// TIA Portal V20 export
TYPE "LBP_typeTMMagazines"
TITLE = Tool management magazines / Magasins de gestion des outils
// User data type to store the magazine data / Type de données utilisateur pour l'enregistrement des données de magasin
   STRUCT
      MaxSpindleNumber : UInt;   // Maximum spindle number / Nombre maximal de broches
      NumberOfMagazines : UInt;   // Number of all magazines including loading and buffer magazines / Nombre total de magasins, y compris les magasins de chargement et de tampon
      Magazines : Array[1..64] of Struct   // All magazines including loading and buffer magazines / Tous les magasins, y compris les magasins de chargement et de tampon
         Number : UInt;   // Magazine number / Numéro de magasin
         "Type" : UInt;   // Magazine type / Type de magasin
         Places : UInt;   // Number of locations in magazine / Nombre d'emplacements dans le magasin
         TMNumber : UInt;   // Tool management number / Numéro de gestion des outils
      END_STRUCT;
   END_STRUCT;
   // // Magazines[2].Number : Magazine number / Numéro de magasin
   // // Magazines[3].Number : Magazine number / Numéro de magasin
   // // Magazines[4].Number : Magazine number / Numéro de magasin
   // // Magazines[5].Number : Magazine number / Numéro de magasin
   // // Magazines[6].Number : Magazine number / Numéro de magasin
   // // Magazines[7].Number : Magazine number / Numéro de magasin
   // // Magazines[8].Number : Magazine number / Numéro de magasin
   // // Magazines[9].Number : Magazine number / Numéro de magasin
   // // Magazines[10].Number : Magazine number / Numéro de magasin
   // // Magazines[11].Number : Magazine number / Numéro de magasin
   // // Magazines[12].Number : Magazine number / Numéro de magasin
   // // Magazines[13].Number : Magazine number / Numéro de magasin
   // // Magazines[14].Number : Magazine number / Numéro de magasin
   // // Magazines[15].Number : Magazine number / Numéro de magasin
   // // Magazines[16].Number : Magazine number / Numéro de magasin
   // // Magazines[17].Number : Magazine number / Numéro de magasin
   // // Magazines[18].Number : Magazine number / Numéro de magasin
   // // Magazines[19].Number : Magazine number / Numéro de magasin
   // // Magazines[20].Number : Magazine number / Numéro de magasin
   // // Magazines[21].Number : Magazine number / Numéro de magasin
   // // Magazines[22].Number : Magazine number / Numéro de magasin
   // // Magazines[23].Number : Magazine number / Numéro de magasin
   // // Magazines[24].Number : Magazine number / Numéro de magasin
   // // Magazines[25].Number : Magazine number / Numéro de magasin
   // // Magazines[26].Number : Magazine number / Numéro de magasin
   // // Magazines[27].Number : Magazine number / Numéro de magasin
   // // Magazines[28].Number : Magazine number / Numéro de magasin
   // // Magazines[29].Number : Magazine number / Numéro de magasin
   // // Magazines[30].Number : Magazine number / Numéro de magasin
   // // Magazines[31].Number : Magazine number / Numéro de magasin
   // // Magazines[32].Number : Magazine number / Numéro de magasin
   // // Magazines[33].Number : Magazine number / Numéro de magasin
   // // Magazines[34].Number : Magazine number / Numéro de magasin
   // // Magazines[35].Number : Magazine number / Numéro de magasin
   // // Magazines[36].Number : Magazine number / Numéro de magasin
   // // Magazines[37].Number : Magazine number / Numéro de magasin
   // // Magazines[38].Number : Magazine number / Numéro de magasin
   // // Magazines[39].Number : Magazine number / Numéro de magasin
   // // Magazines[40].Number : Magazine number / Numéro de magasin
   // // Magazines[41].Number : Magazine number / Numéro de magasin
   // // Magazines[42].Number : Magazine number / Numéro de magasin
   // // Magazines[43].Number : Magazine number / Numéro de magasin
   // // Magazines[44].Number : Magazine number / Numéro de magasin
   // // Magazines[45].Number : Magazine number / Numéro de magasin
   // // Magazines[46].Number : Magazine number / Numéro de magasin
   // // Magazines[47].Number : Magazine number / Numéro de magasin
   // // Magazines[48].Number : Magazine number / Numéro de magasin
   // // Magazines[49].Number : Magazine number / Numéro de magasin
   // // Magazines[50].Number : Magazine number / Numéro de magasin
   // // Magazines[51].Number : Magazine number / Numéro de magasin
   // // Magazines[52].Number : Magazine number / Numéro de magasin
   // // Magazines[53].Number : Magazine number / Numéro de magasin
   // // Magazines[54].Number : Magazine number / Numéro de magasin
   // // Magazines[55].Number : Magazine number / Numéro de magasin
   // // Magazines[56].Number : Magazine number / Numéro de magasin
   // // Magazines[57].Number : Magazine number / Numéro de magasin
   // // Magazines[58].Number : Magazine number / Numéro de magasin
   // // Magazines[59].Number : Magazine number / Numéro de magasin
   // // Magazines[60].Number : Magazine number / Numéro de magasin
   // // Magazines[61].Number : Magazine number / Numéro de magasin
   // // Magazines[62].Number : Magazine number / Numéro de magasin
   // // Magazines[63].Number : Magazine number / Numéro de magasin
   // // Magazines[64].Number : Magazine number / Numéro de magasin
   // // Magazines[2]."Type" : Magazine type / Type de magasin
   // // Magazines[3]."Type" : Magazine type / Type de magasin
   // // Magazines[4]."Type" : Magazine type / Type de magasin
   // // Magazines[5]."Type" : Magazine type / Type de magasin
   // // Magazines[6]."Type" : Magazine type / Type de magasin
   // // Magazines[7]."Type" : Magazine type / Type de magasin
   // // Magazines[8]."Type" : Magazine type / Type de magasin
   // // Magazines[9]."Type" : Magazine type / Type de magasin
   // // Magazines[10]."Type" : Magazine type / Type de magasin
   // // Magazines[11]."Type" : Magazine type / Type de magasin
   // // Magazines[12]."Type" : Magazine type / Type de magasin
   // // Magazines[13]."Type" : Magazine type / Type de magasin
   // // Magazines[14]."Type" : Magazine type / Type de magasin
   // // Magazines[15]."Type" : Magazine type / Type de magasin
   // // Magazines[16]."Type" : Magazine type / Type de magasin
   // // Magazines[17]."Type" : Magazine type / Type de magasin
   // // Magazines[18]."Type" : Magazine type / Type de magasin
   // // Magazines[19]."Type" : Magazine type / Type de magasin
   // // Magazines[20]."Type" : Magazine type / Type de magasin
   // // Magazines[21]."Type" : Magazine type / Type de magasin
   // // Magazines[22]."Type" : Magazine type / Type de magasin
   // // Magazines[23]."Type" : Magazine type / Type de magasin
   // // Magazines[24]."Type" : Magazine type / Type de magasin
   // // Magazines[25]."Type" : Magazine type / Type de magasin
   // // Magazines[26]."Type" : Magazine type / Type de magasin
   // // Magazines[27]."Type" : Magazine type / Type de magasin
   // // Magazines[28]."Type" : Magazine type / Type de magasin
   // // Magazines[29]."Type" : Magazine type / Type de magasin
   // // Magazines[30]."Type" : Magazine type / Type de magasin
   // // Magazines[31]."Type" : Magazine type / Type de magasin
   // // Magazines[32]."Type" : Magazine type / Type de magasin
   // // Magazines[33]."Type" : Magazine type / Type de magasin
   // // Magazines[34]."Type" : Magazine type / Type de magasin
   // // Magazines[35]."Type" : Magazine type / Type de magasin
   // // Magazines[36]."Type" : Magazine type / Type de magasin
   // // Magazines[37]."Type" : Magazine type / Type de magasin
   // // Magazines[38]."Type" : Magazine type / Type de magasin
   // // Magazines[39]."Type" : Magazine type / Type de magasin
   // // Magazines[40]."Type" : Magazine type / Type de magasin
   // // Magazines[41]."Type" : Magazine type / Type de magasin
   // // Magazines[42]."Type" : Magazine type / Type de magasin
   // // Magazines[43]."Type" : Magazine type / Type de magasin
   // // Magazines[44]."Type" : Magazine type / Type de magasin
   // // Magazines[45]."Type" : Magazine type / Type de magasin
   // // Magazines[46]."Type" : Magazine type / Type de magasin
   // // Magazines[47]."Type" : Magazine type / Type de magasin
   // // Magazines[48]."Type" : Magazine type / Type de magasin
   // // Magazines[49]."Type" : Magazine type / Type de magasin
   // // Magazines[50]."Type" : Magazine type / Type de magasin
   // // Magazines[51]."Type" : Magazine type / Type de magasin
   // // Magazines[52]."Type" : Magazine type / Type de magasin
   // // Magazines[53]."Type" : Magazine type / Type de magasin
   // // Magazines[54]."Type" : Magazine type / Type de magasin
   // // Magazines[55]."Type" : Magazine type / Type de magasin
   // // Magazines[56]."Type" : Magazine type / Type de magasin
   // // Magazines[57]."Type" : Magazine type / Type de magasin
   // // Magazines[58]."Type" : Magazine type / Type de magasin
   // // Magazines[59]."Type" : Magazine type / Type de magasin
   // // Magazines[60]."Type" : Magazine type / Type de magasin
   // // Magazines[61]."Type" : Magazine type / Type de magasin
   // // Magazines[62]."Type" : Magazine type / Type de magasin
   // // Magazines[63]."Type" : Magazine type / Type de magasin
   // // Magazines[64]."Type" : Magazine type / Type de magasin
   // // Magazines[2].Places : Number of locations in magazine / Nombre d'emplacements dans le magasin
   // // Magazines[3].Places : Number of locations in magazine / Nombre d'emplacements dans le magasin
   // // Magazines[4].Places : Number of locations in magazine / Nombre d'emplacements dans le magasin
   // // Magazines[5].Places : Number of locations in magazine / Nombre d'emplacements dans le magasin
   // // Magazines[6].Places : Number of locations in magazine / Nombre d'emplacements dans le magasin
   // // Magazines[7].Places : Number of locations in magazine / Nombre d'emplacements dans le magasin
   // // Magazines[8].Places : Number of locations in magazine / Nombre d'emplacements dans le magasin
   // // Magazines[9].Places : Number of locations in magazine / Nombre d'emplacements dans le magasin
   // // Magazines[10].Places : Number of locations in magazine / Nombre d'emplacements dans le magasin
   // // Magazines[11].Places : Number of locations in magazine / Nombre d'emplacements dans le magasin
   // // Magazines[12].Places : Number of locations in magazine / Nombre d'emplacements dans le magasin
   // // Magazines[13].Places : Number of locations in magazine / Nombre d'emplacements dans le magasin
   // // Magazines[14].Places : Number of locations in magazine / Nombre d'emplacements dans le magasin
   // // Magazines[15].Places : Number of locations in magazine / Nombre d'emplacements dans le magasin
   // // Magazines[16].Places : Number of locations in magazine / Nombre d'emplacements dans le magasin
   // // Magazines[17].Places : Number of locations in magazine / Nombre d'emplacements dans le magasin
   // // Magazines[18].Places : Number of locations in magazine / Nombre d'emplacements dans le magasin
   // // Magazines[19].Places : Number of locations in magazine / Nombre d'emplacements dans le magasin
   // // Magazines[20].Places : Number of locations in magazine / Nombre d'emplacements dans le magasin
   // // Magazines[21].Places : Number of locations in magazine / Nombre d'emplacements dans le magasin
   // // Magazines[22].Places : Number of locations in magazine / Nombre d'emplacements dans le magasin
   // // Magazines[23].Places : Number of locations in magazine / Nombre d'emplacements dans le magasin
   // // Magazines[24].Places : Number of locations in magazine / Nombre d'emplacements dans le magasin
   // // Magazines[25].Places : Number of locations in magazine / Nombre d'emplacements dans le magasin
   // // Magazines[26].Places : Number of locations in magazine / Nombre d'emplacements dans le magasin
   // // Magazines[27].Places : Number of locations in magazine / Nombre d'emplacements dans le magasin
   // // Magazines[28].Places : Number of locations in magazine / Nombre d'emplacements dans le magasin
   // // Magazines[29].Places : Number of locations in magazine / Nombre d'emplacements dans le magasin
   // // Magazines[30].Places : Number of locations in magazine / Nombre d'emplacements dans le magasin
   // // Magazines[31].Places : Number of locations in magazine / Nombre d'emplacements dans le magasin
   // // Magazines[32].Places : Number of locations in magazine / Nombre d'emplacements dans le magasin
   // // Magazines[33].Places : Number of locations in magazine / Nombre d'emplacements dans le magasin
   // // Magazines[34].Places : Number of locations in magazine / Nombre d'emplacements dans le magasin
   // // Magazines[35].Places : Number of locations in magazine / Nombre d'emplacements dans le magasin
   // // Magazines[36].Places : Number of locations in magazine / Nombre d'emplacements dans le magasin
   // // Magazines[37].Places : Number of locations in magazine / Nombre d'emplacements dans le magasin
   // // Magazines[38].Places : Number of locations in magazine / Nombre d'emplacements dans le magasin
   // // Magazines[39].Places : Number of locations in magazine / Nombre d'emplacements dans le magasin
   // // Magazines[40].Places : Number of locations in magazine / Nombre d'emplacements dans le magasin
   // // Magazines[41].Places : Number of locations in magazine / Nombre d'emplacements dans le magasin
   // // Magazines[42].Places : Number of locations in magazine / Nombre d'emplacements dans le magasin
   // // Magazines[43].Places : Number of locations in magazine / Nombre d'emplacements dans le magasin
   // // Magazines[44].Places : Number of locations in magazine / Nombre d'emplacements dans le magasin
   // // Magazines[45].Places : Number of locations in magazine / Nombre d'emplacements dans le magasin
   // // Magazines[46].Places : Number of locations in magazine / Nombre d'emplacements dans le magasin
   // // Magazines[47].Places : Number of locations in magazine / Nombre d'emplacements dans le magasin
   // // Magazines[48].Places : Number of locations in magazine / Nombre d'emplacements dans le magasin
   // // Magazines[49].Places : Number of locations in magazine / Nombre d'emplacements dans le magasin
   // // Magazines[50].Places : Number of locations in magazine / Nombre d'emplacements dans le magasin
   // // Magazines[51].Places : Number of locations in magazine / Nombre d'emplacements dans le magasin
   // // Magazines[52].Places : Number of locations in magazine / Nombre d'emplacements dans le magasin
   // // Magazines[53].Places : Number of locations in magazine / Nombre d'emplacements dans le magasin
   // // Magazines[54].Places : Number of locations in magazine / Nombre d'emplacements dans le magasin
   // // Magazines[55].Places : Number of locations in magazine / Nombre d'emplacements dans le magasin
   // // Magazines[56].Places : Number of locations in magazine / Nombre d'emplacements dans le magasin
   // // Magazines[57].Places : Number of locations in magazine / Nombre d'emplacements dans le magasin
   // // Magazines[58].Places : Number of locations in magazine / Nombre d'emplacements dans le magasin
   // // Magazines[59].Places : Number of locations in magazine / Nombre d'emplacements dans le magasin
   // // Magazines[60].Places : Number of locations in magazine / Nombre d'emplacements dans le magasin
   // // Magazines[61].Places : Number of locations in magazine / Nombre d'emplacements dans le magasin
   // // Magazines[62].Places : Number of locations in magazine / Nombre d'emplacements dans le magasin
   // // Magazines[63].Places : Number of locations in magazine / Nombre d'emplacements dans le magasin
   // // Magazines[64].Places : Number of locations in magazine / Nombre d'emplacements dans le magasin
   // // Magazines[2].TMNumber : Tool management number / Numéro de gestion des outils
   // // Magazines[3].TMNumber : Tool management number / Numéro de gestion des outils
   // // Magazines[4].TMNumber : Tool management number / Numéro de gestion des outils
   // // Magazines[5].TMNumber : Tool management number / Numéro de gestion des outils
   // // Magazines[6].TMNumber : Tool management number / Numéro de gestion des outils
   // // Magazines[7].TMNumber : Tool management number / Numéro de gestion des outils
   // // Magazines[8].TMNumber : Tool management number / Numéro de gestion des outils
   // // Magazines[9].TMNumber : Tool management number / Numéro de gestion des outils
   // // Magazines[10].TMNumber : Tool management number / Numéro de gestion des outils
   // // Magazines[11].TMNumber : Tool management number / Numéro de gestion des outils
   // // Magazines[12].TMNumber : Tool management number / Numéro de gestion des outils
   // // Magazines[13].TMNumber : Tool management number / Numéro de gestion des outils
   // // Magazines[14].TMNumber : Tool management number / Numéro de gestion des outils
   // // Magazines[15].TMNumber : Tool management number / Numéro de gestion des outils
   // // Magazines[16].TMNumber : Tool management number / Numéro de gestion des outils
   // // Magazines[17].TMNumber : Tool management number / Numéro de gestion des outils
   // // Magazines[18].TMNumber : Tool management number / Numéro de gestion des outils
   // // Magazines[19].TMNumber : Tool management number / Numéro de gestion des outils
   // // Magazines[20].TMNumber : Tool management number / Numéro de gestion des outils
   // // Magazines[21].TMNumber : Tool management number / Numéro de gestion des outils
   // // Magazines[22].TMNumber : Tool management number / Numéro de gestion des outils
   // // Magazines[23].TMNumber : Tool management number / Numéro de gestion des outils
   // // Magazines[24].TMNumber : Tool management number / Numéro de gestion des outils
   // // Magazines[25].TMNumber : Tool management number / Numéro de gestion des outils
   // // Magazines[26].TMNumber : Tool management number / Numéro de gestion des outils
   // // Magazines[27].TMNumber : Tool management number / Numéro de gestion des outils
   // // Magazines[28].TMNumber : Tool management number / Numéro de gestion des outils
   // // Magazines[29].TMNumber : Tool management number / Numéro de gestion des outils
   // // Magazines[30].TMNumber : Tool management number / Numéro de gestion des outils
   // // Magazines[31].TMNumber : Tool management number / Numéro de gestion des outils
   // // Magazines[32].TMNumber : Tool management number / Numéro de gestion des outils
   // // Magazines[33].TMNumber : Tool management number / Numéro de gestion des outils
   // // Magazines[34].TMNumber : Tool management number / Numéro de gestion des outils
   // // Magazines[35].TMNumber : Tool management number / Numéro de gestion des outils
   // // Magazines[36].TMNumber : Tool management number / Numéro de gestion des outils
   // // Magazines[37].TMNumber : Tool management number / Numéro de gestion des outils
   // // Magazines[38].TMNumber : Tool management number / Numéro de gestion des outils
   // // Magazines[39].TMNumber : Tool management number / Numéro de gestion des outils
   // // Magazines[40].TMNumber : Tool management number / Numéro de gestion des outils
   // // Magazines[41].TMNumber : Tool management number / Numéro de gestion des outils
   // // Magazines[42].TMNumber : Tool management number / Numéro de gestion des outils
   // // Magazines[43].TMNumber : Tool management number / Numéro de gestion des outils
   // // Magazines[44].TMNumber : Tool management number / Numéro de gestion des outils
   // // Magazines[45].TMNumber : Tool management number / Numéro de gestion des outils
   // // Magazines[46].TMNumber : Tool management number / Numéro de gestion des outils
   // // Magazines[47].TMNumber : Tool management number / Numéro de gestion des outils
   // // Magazines[48].TMNumber : Tool management number / Numéro de gestion des outils
   // // Magazines[49].TMNumber : Tool management number / Numéro de gestion des outils
   // // Magazines[50].TMNumber : Tool management number / Numéro de gestion des outils
   // // Magazines[51].TMNumber : Tool management number / Numéro de gestion des outils
   // // Magazines[52].TMNumber : Tool management number / Numéro de gestion des outils
   // // Magazines[53].TMNumber : Tool management number / Numéro de gestion des outils
   // // Magazines[54].TMNumber : Tool management number / Numéro de gestion des outils
   // // Magazines[55].TMNumber : Tool management number / Numéro de gestion des outils
   // // Magazines[56].TMNumber : Tool management number / Numéro de gestion des outils
   // // Magazines[57].TMNumber : Tool management number / Numéro de gestion des outils
   // // Magazines[58].TMNumber : Tool management number / Numéro de gestion des outils
   // // Magazines[59].TMNumber : Tool management number / Numéro de gestion des outils
   // // Magazines[60].TMNumber : Tool management number / Numéro de gestion des outils
   // // Magazines[61].TMNumber : Tool management number / Numéro de gestion des outils
   // // Magazines[62].TMNumber : Tool management number / Numéro de gestion des outils
   // // Magazines[63].TMNumber : Tool management number / Numéro de gestion des outils
   // // Magazines[64].TMNumber : Tool management number / Numéro de gestion des outils
   // // Magazines[1] : All magazines including loading and buffer magazines / Tous les magasins, y compris les magasins de chargement et de tampon
   // // Magazines[2] : All magazines including loading and buffer magazines / Tous les magasins, y compris les magasins de chargement et de tampon
   // // Magazines[3] : All magazines including loading and buffer magazines / Tous les magasins, y compris les magasins de chargement et de tampon
   // // Magazines[4] : All magazines including loading and buffer magazines / Tous les magasins, y compris les magasins de chargement et de tampon
   // // Magazines[5] : All magazines including loading and buffer magazines / Tous les magasins, y compris les magasins de chargement et de tampon
   // // Magazines[6] : All magazines including loading and buffer magazines / Tous les magasins, y compris les magasins de chargement et de tampon
   // // Magazines[7] : All magazines including loading and buffer magazines / Tous les magasins, y compris les magasins de chargement et de tampon
   // // Magazines[8] : All magazines including loading and buffer magazines / Tous les magasins, y compris les magasins de chargement et de tampon
   // // Magazines[9] : All magazines including loading and buffer magazines / Tous les magasins, y compris les magasins de chargement et de tampon
   // // Magazines[10] : All magazines including loading and buffer magazines / Tous les magasins, y compris les magasins de chargement et de tampon
   // // Magazines[11] : All magazines including loading and buffer magazines / Tous les magasins, y compris les magasins de chargement et de tampon
   // // Magazines[12] : All magazines including loading and buffer magazines / Tous les magasins, y compris les magasins de chargement et de tampon
   // // Magazines[13] : All magazines including loading and buffer magazines / Tous les magasins, y compris les magasins de chargement et de tampon
   // // Magazines[14] : All magazines including loading and buffer magazines / Tous les magasins, y compris les magasins de chargement et de tampon
   // // Magazines[15] : All magazines including loading and buffer magazines / Tous les magasins, y compris les magasins de chargement et de tampon
   // // Magazines[16] : All magazines including loading and buffer magazines / Tous les magasins, y compris les magasins de chargement et de tampon
   // // Magazines[17] : All magazines including loading and buffer magazines / Tous les magasins, y compris les magasins de chargement et de tampon
   // // Magazines[18] : All magazines including loading and buffer magazines / Tous les magasins, y compris les magasins de chargement et de tampon
   // // Magazines[19] : All magazines including loading and buffer magazines / Tous les magasins, y compris les magasins de chargement et de tampon
   // // Magazines[20] : All magazines including loading and buffer magazines / Tous les magasins, y compris les magasins de chargement et de tampon
   // // Magazines[21] : All magazines including loading and buffer magazines / Tous les magasins, y compris les magasins de chargement et de tampon
   // // Magazines[22] : All magazines including loading and buffer magazines / Tous les magasins, y compris les magasins de chargement et de tampon
   // // Magazines[23] : All magazines including loading and buffer magazines / Tous les magasins, y compris les magasins de chargement et de tampon
   // // Magazines[24] : All magazines including loading and buffer magazines / Tous les magasins, y compris les magasins de chargement et de tampon
   // // Magazines[25] : All magazines including loading and buffer magazines / Tous les magasins, y compris les magasins de chargement et de tampon
   // // Magazines[26] : All magazines including loading and buffer magazines / Tous les magasins, y compris les magasins de chargement et de tampon
   // // Magazines[27] : All magazines including loading and buffer magazines / Tous les magasins, y compris les magasins de chargement et de tampon
   // // Magazines[28] : All magazines including loading and buffer magazines / Tous les magasins, y compris les magasins de chargement et de tampon
   // // Magazines[29] : All magazines including loading and buffer magazines / Tous les magasins, y compris les magasins de chargement et de tampon
   // // Magazines[30] : All magazines including loading and buffer magazines / Tous les magasins, y compris les magasins de chargement et de tampon
   // // Magazines[31] : All magazines including loading and buffer magazines / Tous les magasins, y compris les magasins de chargement et de tampon
   // // Magazines[32] : All magazines including loading and buffer magazines / Tous les magasins, y compris les magasins de chargement et de tampon
   // // Magazines[33] : All magazines including loading and buffer magazines / Tous les magasins, y compris les magasins de chargement et de tampon
   // // Magazines[34] : All magazines including loading and buffer magazines / Tous les magasins, y compris les magasins de chargement et de tampon
   // // Magazines[35] : All magazines including loading and buffer magazines / Tous les magasins, y compris les magasins de chargement et de tampon
   // // Magazines[36] : All magazines including loading and buffer magazines / Tous les magasins, y compris les magasins de chargement et de tampon
   // // Magazines[37] : All magazines including loading and buffer magazines / Tous les magasins, y compris les magasins de chargement et de tampon
   // // Magazines[38] : All magazines including loading and buffer magazines / Tous les magasins, y compris les magasins de chargement et de tampon
   // // Magazines[39] : All magazines including loading and buffer magazines / Tous les magasins, y compris les magasins de chargement et de tampon
   // // Magazines[40] : All magazines including loading and buffer magazines / Tous les magasins, y compris les magasins de chargement et de tampon
   // // Magazines[41] : All magazines including loading and buffer magazines / Tous les magasins, y compris les magasins de chargement et de tampon
   // // Magazines[42] : All magazines including loading and buffer magazines / Tous les magasins, y compris les magasins de chargement et de tampon
   // // Magazines[43] : All magazines including loading and buffer magazines / Tous les magasins, y compris les magasins de chargement et de tampon
   // // Magazines[44] : All magazines including loading and buffer magazines / Tous les magasins, y compris les magasins de chargement et de tampon
   // // Magazines[45] : All magazines including loading and buffer magazines / Tous les magasins, y compris les magasins de chargement et de tampon
   // // Magazines[46] : All magazines including loading and buffer magazines / Tous les magasins, y compris les magasins de chargement et de tampon
   // // Magazines[47] : All magazines including loading and buffer magazines / Tous les magasins, y compris les magasins de chargement et de tampon
   // // Magazines[48] : All magazines including loading and buffer magazines / Tous les magasins, y compris les magasins de chargement et de tampon
   // // Magazines[49] : All magazines including loading and buffer magazines / Tous les magasins, y compris les magasins de chargement et de tampon
   // // Magazines[50] : All magazines including loading and buffer magazines / Tous les magasins, y compris les magasins de chargement et de tampon
   // // Magazines[51] : All magazines including loading and buffer magazines / Tous les magasins, y compris les magasins de chargement et de tampon
   // // Magazines[52] : All magazines including loading and buffer magazines / Tous les magasins, y compris les magasins de chargement et de tampon
   // // Magazines[53] : All magazines including loading and buffer magazines / Tous les magasins, y compris les magasins de chargement et de tampon
   // // Magazines[54] : All magazines including loading and buffer magazines / Tous les magasins, y compris les magasins de chargement et de tampon
   // // Magazines[55] : All magazines including loading and buffer magazines / Tous les magasins, y compris les magasins de chargement et de tampon
   // // Magazines[56] : All magazines including loading and buffer magazines / Tous les magasins, y compris les magasins de chargement et de tampon
   // // Magazines[57] : All magazines including loading and buffer magazines / Tous les magasins, y compris les magasins de chargement et de tampon
   // // Magazines[58] : All magazines including loading and buffer magazines / Tous les magasins, y compris les magasins de chargement et de tampon
   // // Magazines[59] : All magazines including loading and buffer magazines / Tous les magasins, y compris les magasins de chargement et de tampon
   // // Magazines[60] : All magazines including loading and buffer magazines / Tous les magasins, y compris les magasins de chargement et de tampon
   // // Magazines[61] : All magazines including loading and buffer magazines / Tous les magasins, y compris les magasins de chargement et de tampon
   // // Magazines[62] : All magazines including loading and buffer magazines / Tous les magasins, y compris les magasins de chargement et de tampon
   // // Magazines[63] : All magazines including loading and buffer magazines / Tous les magasins, y compris les magasins de chargement et de tampon
   // // Magazines[64] : All magazines including loading and buffer magazines / Tous les magasins, y compris les magasins de chargement et de tampon
END_TYPE
